// TIA Portal V20 program export: 3 tag tables, 2 data types, 2 data blocks, 7 code blocks (in call order from the OBs), 11 instance data blocks

VAR_GLOBAL   // PLC tag table "Default tag table"
   All_Lamps AT %QB0 : Byte;
   Lamps_On AT %Q5.0 : Bool;
   Light2State AT %M0.0 : Bool;
   Light1State AT %M0.1 : Bool;
   Light3State AT %M0.2 : Bool;
   LightStep AT %MW0 : Int;
   start AT %M2.0 : Bool;
   Elapsed_Time AT %MD4 : Time;
   Lamps AT %MB0 : Byte;
END_VAR

VAR_GLOBAL   // PLC tag table "Inputs"
   "Switch 1 ON" AT %I16.0 : Bool;
   "Switch 2 ON" AT %I16.1 : Bool;
   "Switch 3 ON" AT %I16.2 : Bool;
   "Switch 4 ON" AT %I16.3 : Bool;
   "Switch 5 ON" AT %I16.4 : Bool;
   "Switch 6 ON" AT %I16.5 : Bool;
   "Switch 7 ON" AT %I16.6 : Bool;
   "Switch 8 ON" AT %I16.7 : Bool;
   "Byte 1 ON" AT %IB1 : Byte;
   Here_is_a_word AT %IW2 : Word;
END_VAR

VAR_GLOBAL   // PLC tag table "Outputs"
   "Lamp 1 ON" AT %Q0.0 : Bool;
   "Lamp 2 ON" AT %Q0.1 : Bool;
   "Lamp 3 ON" AT %Q0.2 : Bool;
   "Lamp 4 ON" AT %Q0.3 : Bool;
   "Lamp 5 ON" AT %Q0.4 : Bool;
   "Lamp 6 ON" AT %Q0.5 : Bool;
   "Lamp 7 ON" AT %Q0.6 : Bool;
   "Lamp 8 ON" AT %Q0.7 : Bool;
   I_am_a_double_integer AT %QD1 : DInt;
END_VAR

TYPE "Equipment"
   STRUCT
      "type" : Int;
      commandOn : Bool;
      commandOff : Bool;
      feedbackOn : Bool;
      feedbackOff : Bool;
      isFaulty : Bool;
      isProcessFinished : Bool;
   END_STRUCT;
END_TYPE

TYPE "Tank"
   STRUCT
      isTankFull : Bool;
      tankLevel : Int;
      isEmpty : Bool;
      "type" : Bool;
   END_STRUCT;
END_TYPE

DATA_BLOCK "Global DB"   // DB7
{ S7_Optimized_Access := 'TRUE' }
// stored: MemoryReserve 100
   VAR
      Valve1 : "Equipment";
      Valve2 { S7_SetPoint := 'True'} : "Equipment";
      Valve3 { S7_SetPoint := 'True'} : "Equipment";
      Heater { S7_SetPoint := 'True'} : "Equipment";
      Mixer { S7_SetPoint := 'True'} : "Equipment";
      Process_Start { S7_SetPoint := 'True'} : Bool;
      Process_Stop : Bool;
      Process_Reset : Bool;
      Process_Step : Int;
      Process_Count : Int;
      isTankHeated : Bool;
      isTankMixed : Bool;
      Tank1 : "Tank";
      Tank2 { S7_SetPoint := 'True'} : "Tank";
      positive_edge { S7_SetPoint := 'True'} : Bool;
      prevLevel : DInt;
   END_VAR
BEGIN
   Heater."type" := 1;
   Mixer."type" := 2;
END_DATA_BLOCK

DATA_BLOCK "DB_Traffic_Lights"   // DB1
{ S7_Optimized_Access := 'TRUE' }
// stored: MemoryReserve 100
   VAR
      Process_Step : Int;
      Process_Start : Bool;
      "Timer" : IEC_TIMER;
      "Counter" { S7_SetPoint := 'True'} : IEC_COUNTER;
   END_VAR
   VAR RETAIN
      Positive_Edge { S7_SetPoint := 'True'} : Bool;
   END_VAR
   VAR
      Timer2 : IEC_TIMER;
   END_VAR
BEGIN
END_DATA_BLOCK

ORGANIZATION_BLOCK "Main"   // OB1, LAD, ProgramCycle
TITLE = "Main Program Sweep (Cycle)"
{ S7_Optimized_Access := 'TRUE' }
// stored: SetENOAutomatically false
   VAR_INPUT
      Initial_Call : Bool;   // Initial call of this OB
      Remanence : Bool;   // =True, if remanent data are available
   END_VAR
BEGIN

REGION Network 1
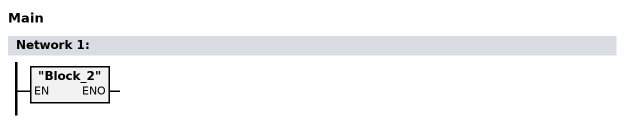
   RUNG wire#powerrail
      "Block_2"()
   END_RUNG
   // the same network as SCL:
   "Block_2"();
END_REGION
END_ORGANIZATION_BLOCK

FUNCTION "Block_2" : Void   // FC2, LAD
{ S7_Optimized_Access := 'TRUE' }
// stored: SetENOAutomatically false
   VAR_TEMP   // added for the SCL form of the ladder/FBD networks
      _w1 : Bool;
   END_VAR
BEGIN

REGION Network 1
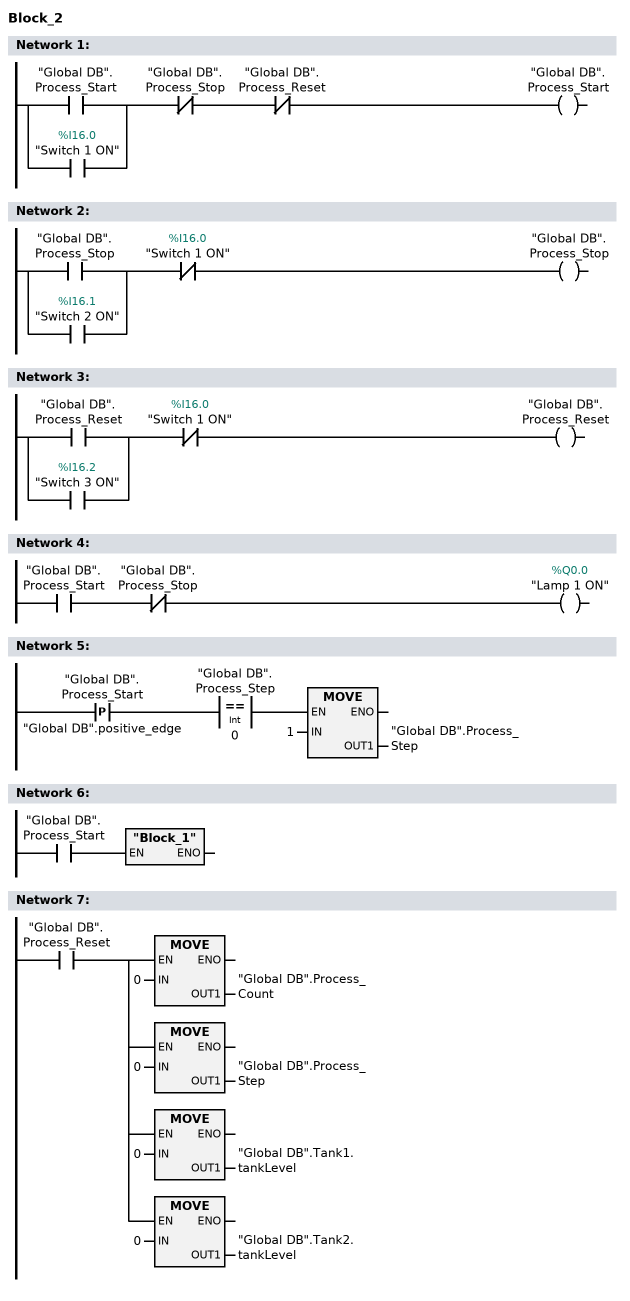
   RUNG wire#powerrail
      Contact( "Global DB".Process_Start )
      wire#w1
      I_Contact( "Global DB".Process_Stop )
      I_Contact( "Global DB".Process_Reset )
      Coil( "Global DB".Process_Start )
   END_RUNG
   RUNG wire#powerrail
      Contact( "Switch 1 ON" )
   END_RUNG wire#w1
   // the same network as SCL:
   "Global DB".Process_Start := ("Global DB".Process_Start OR "Switch 1 ON") AND NOT "Global DB".Process_Stop AND NOT "Global DB".Process_Reset;
END_REGION

REGION Network 2
   RUNG wire#powerrail
      Contact( "Global DB".Process_Stop )
      wire#w1
      I_Contact( "Switch 1 ON" )
      Coil( "Global DB".Process_Stop )
   END_RUNG
   RUNG wire#powerrail
      Contact( "Switch 2 ON" )
   END_RUNG wire#w1
   // the same network as SCL:
   "Global DB".Process_Stop := ("Global DB".Process_Stop OR "Switch 2 ON") AND NOT "Switch 1 ON";
END_REGION

REGION Network 3
   RUNG wire#powerrail
      Contact( "Global DB".Process_Reset )
      wire#w1
      I_Contact( "Switch 1 ON" )
      Coil( "Global DB".Process_Reset )
   END_RUNG
   RUNG wire#powerrail
      Contact( "Switch 3 ON" )
   END_RUNG wire#w1
   // the same network as SCL:
   "Global DB".Process_Reset := ("Global DB".Process_Reset OR "Switch 3 ON") AND NOT "Switch 1 ON";
END_REGION

REGION Network 4
   RUNG wire#powerrail
      Contact( "Global DB".Process_Start )
      I_Contact( "Global DB".Process_Stop )
      Coil( "Lamp 1 ON" )
   END_RUNG
   // the same network as SCL:
   "Lamp 1 ON" := "Global DB".Process_Start AND NOT "Global DB".Process_Stop;
END_REGION

REGION Network 5
   RUNG wire#powerrail
      P_Contact(operand := "Global DB".Process_Start, bit := "Global DB".positive_edge)
      { S7_Templates := "SrcType := Int" } EQ_Contact(in1 := "Global DB".Process_Step, in2 := 0)
      Move(in := 1, out1 => "Global DB".Process_Step)
   END_RUNG
   // the same network as SCL:
   #_w1 := "Global DB".Process_Start AND NOT "Global DB".positive_edge;   // rising edge of "Global DB".Process_Start
   "Global DB".positive_edge := "Global DB".Process_Start;
   IF #_w1 AND ("Global DB".Process_Step = 0) THEN "Global DB".Process_Step := 1; END_IF;
END_REGION

REGION Network 6
   RUNG wire#powerrail
      Contact( "Global DB".Process_Start )
      "Block_1"()
   END_RUNG
   // the same network as SCL:
   IF "Global DB".Process_Start THEN "Block_1"(); END_IF;
END_REGION

REGION Network 7
   RUNG wire#powerrail
      Contact( "Global DB".Process_Reset )
      wire#w1
      Move(in := 0, out1 => "Global DB".Process_Count)
   END_RUNG
   RUNG wire#w1
      Move(in := 0, out1 => "Global DB".Process_Step)
   END_RUNG
   RUNG wire#w1
      Move(in := 0, out1 => "Global DB".Tank1.tankLevel)
   END_RUNG
   RUNG wire#w1
      Move(in := 0, out1 => "Global DB".Tank2.tankLevel)
   END_RUNG
   // the same network as SCL:
   IF "Global DB".Process_Reset THEN
       "Global DB".Process_Count := 0;
       "Global DB".Process_Step := 0;
       "Global DB".Tank1.tankLevel := 0;
       "Global DB".Tank2.tankLevel := 0;
   END_IF;
END_REGION
END_FUNCTION

FUNCTION "Block_1" : Void
{ S7_Optimized_Access := 'TRUE' }
VERSION : 0.1
   VAR_TEMP 
      prevTankLevel : DInt;
   END_VAR


BEGIN
	
	CASE "Global DB".Process_Step OF
	        
	    1:
	        
	        "Block_3"(eqp := "Global DB".Valve1,
	                  timer := "IEC_Timer_0_DB_4",
	                  tank := "Global DB".Tank1);
	      
	        
	        ;
	        
	        
	    2:
	        
	        "Block_3"(eqp := "Global DB".Heater,
	                  timer := "IEC_Timer_0_DB_5",
	                  tank := "Global DB".Tank1);
	        ;
	        
	        
	    3:
	        "Block_3"(eqp := "Global DB".Mixer,
	                  timer := "IEC_Timer_0_DB_6",
	                  tank := "Global DB".Tank1);
	        ;
	        
	        
	    4:
	 
	        IF ("Global DB".Process_Count < 5) THEN
	            
	            
	            
	            "Global DB".Tank2.tankLevel := "Global DB".prevLevel + (DINT_TO_REAL(TIME_TO_DINT("IEC_Timer_0_DB_7".ET)) / 250.0);
	            "Global DB".Tank1.tankLevel := 100 - DINT_TO_REAL(TIME_TO_DINT("IEC_Timer_0_DB_7".ET)) / 50.0;
	            
	            
	            IF ("IEC_Timer_0_DB_7".Q) THEN
	                
	                
	                "Global DB".prevLevel := "Global DB".Tank2.tankLevel;
	                IF ("Global DB".Tank2.isTankFull) THEN
	                    "Global DB".Process_Step := 5;
	                    "Global DB".Process_Count := 0;
	                ELSE
	                    "Global DB".Process_Count += 1;
	                    "Global DB".Process_Step := 1;
	                END_IF;
	                
	            END_IF;
	            
	            
	        END_IF;
	        
	     5:
	
	         "Global DB".Tank2.tankLevel := 100 - DINT_TO_REAL(TIME_TO_DINT("IEC_Timer_0_DB_8".ET))/ 50.0;
	         
	         IF("IEC_Timer_0_DB_8".Q) THEN
	         "Global DB".Process_Step := 1;
	         "Global DB".prevLevel := 0;
	         
	        END_IF
	         
	         ;
	        
	        
	        
	END_CASE;
	
	"IEC_Timer_0_DB_7".TON(IN := "Global DB".Process_Step = 4,
	                       PT := T#5s);
	
	"IEC_Timer_0_DB_8".TON(IN := "Global DB".Process_Step = 5,
	                       PT := T#5s);
	
	IF ("Global DB".Tank1.tankLevel = 100) THEN
	    "Global DB".Tank1.isTankFull := TRUE
	    ;
	ELSE
	    "Global DB".Tank1.isTankFull := FALSE;
	    
	END_IF;
	
	IF ("Global DB".Tank2.tankLevel = 100) THEN
	    "Global DB".Tank2.isTankFull := TRUE
	    ;
	ELSE
	    "Global DB".Tank2.isTankFull := FALSE;
	    
	END_IF;
END_FUNCTION

FUNCTION "Block_3" : Void
{ S7_Optimized_Access := 'TRUE' }
VERSION : 0.1
   VAR_IN_OUT 
      eqp : "Equipment";
      "timer" {InstructionName := 'IEC_TIMER'; LibVersion := '1.0'} : IEC_TIMER;
      tank : "Tank";
   END_VAR

   VAR_TEMP 
      isNotTank : Bool;
      currentStep : Int;
      currentStepOld : Int;
      isStepDifferent : Bool;
   END_VAR


BEGIN
	
	#eqp.commandOn := TRUE;
	
	
	    
	"IEC_Timer_0_DB_4".TON(
	                       IN := ("Global DB".Process_Step = 1),
	                       PT := T#5s
	                       
	);
	
	"IEC_Timer_0_DB_5".TON(
	                       IN := ("Global DB".Process_Step = 2),
	                       PT := T#5s
	                       
	);
	
	
	
	
	
	
	"IEC_Timer_0_DB_6".TON(
	                       IN := ("Global DB".Process_Step = 3),
	                       PT := T#5s
	                       
	);
	
	
	  
	    CASE #eqp.type OF
	        0:
	            #tank.tankLevel := DINT_TO_REAL(TIME_TO_DINT(#timer.ET)) / 50.0;
	            
	        1..2:
	            #eqp.isProcessFinished := TRUE;
	            
	            
	    END_CASE;
	    
	
	    IF ( #timer.Q) THEN
	        #eqp.commandOn := FALSE;
	        #eqp.commandOff := TRUE;
	        "Global DB".Process_Step += 1
	        ;
	    END_IF;
	    
	 
END_FUNCTION

FUNCTION_BLOCK "FC_Traffic_Lights"   // FB1, LAD
{ S7_Optimized_Access := 'TRUE' }
// stored: MemoryReserve 100, SetENOAutomatically false
   VAR
      "Timer" { S7_SetPoint := 'True'} : TON_TIME;
   END_VAR
   VAR_TEMP   // added for the SCL form of the ladder/FBD networks
      _w1 : Bool;
   END_VAR
BEGIN

REGION Network 1
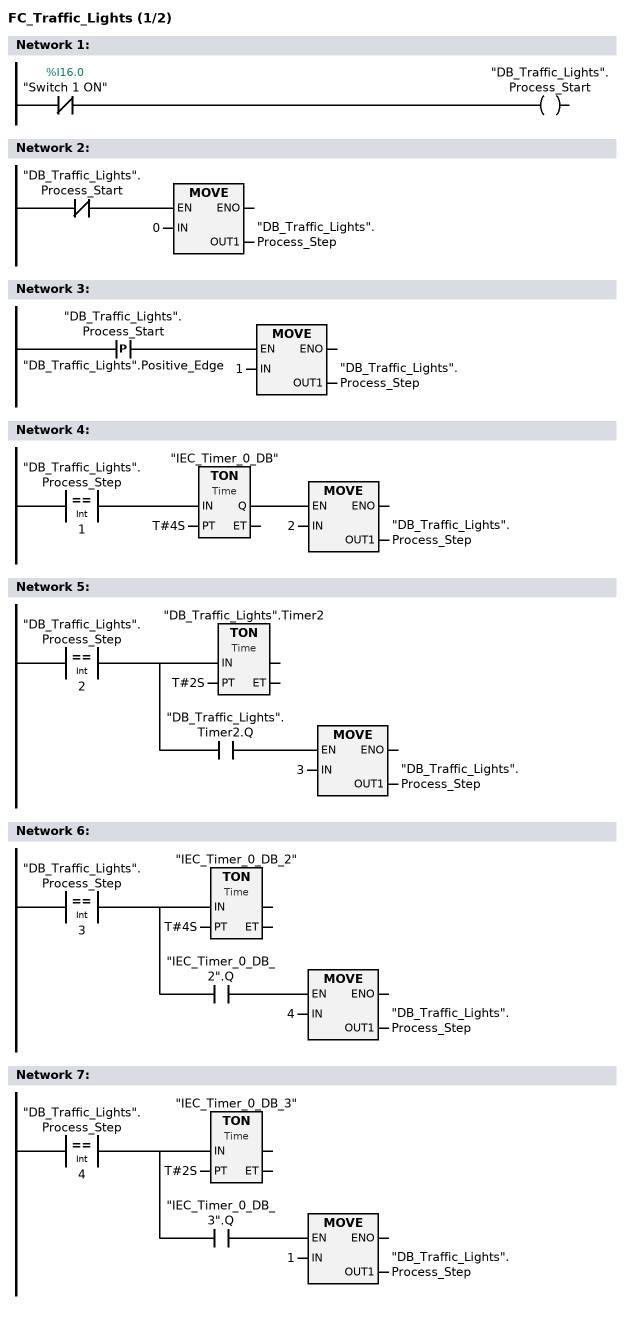
   RUNG wire#powerrail
      I_Contact( "Switch 1 ON" )
      Coil( "DB_Traffic_Lights".Process_Start )
   END_RUNG
   // the same network as SCL:
   "DB_Traffic_Lights".Process_Start := NOT "Switch 1 ON";
END_REGION

REGION Network 2
   RUNG wire#powerrail
      I_Contact( "DB_Traffic_Lights".Process_Start )
      Move(in := 0, out1 => "DB_Traffic_Lights".Process_Step)
   END_RUNG
   // the same network as SCL:
   IF NOT "DB_Traffic_Lights".Process_Start THEN "DB_Traffic_Lights".Process_Step := 0; END_IF;
END_REGION

REGION Network 3
   RUNG wire#powerrail
      P_Contact(operand := "DB_Traffic_Lights".Process_Start, bit := "DB_Traffic_Lights".Positive_Edge)
      Move(in := 1, out1 => "DB_Traffic_Lights".Process_Step)
   END_RUNG
   // the same network as SCL:
   #_w1 := "DB_Traffic_Lights".Process_Start AND NOT "DB_Traffic_Lights".Positive_Edge;   // rising edge of "DB_Traffic_Lights".Process_Start
   "DB_Traffic_Lights".Positive_Edge := "DB_Traffic_Lights".Process_Start;
   IF #_w1 THEN "DB_Traffic_Lights".Process_Step := 1; END_IF;
END_REGION

REGION Network 4
   RUNG wire#powerrail
      { S7_Templates := "SrcType := Int" } EQ_Contact(in1 := "DB_Traffic_Lights".Process_Step, in2 := 1)
      { S7_Templates := "time_type := Time" } "IEC_Timer_0_DB".TON(pt := T#4S, et =>)
      Move(in := 2, out1 => "DB_Traffic_Lights".Process_Step)
   END_RUNG
   // the same network as SCL:
   "IEC_Timer_0_DB".TON(IN := "DB_Traffic_Lights".Process_Step = 1, PT := T#4S);
   IF "IEC_Timer_0_DB".Q THEN "DB_Traffic_Lights".Process_Step := 2; END_IF;
END_REGION

REGION Network 5
   RUNG wire#powerrail
      { S7_Templates := "SrcType := Int" } EQ_Contact(in1 := "DB_Traffic_Lights".Process_Step, in2 := 2)
      wire#w1
      { S7_Templates := "time_type := Time" } "DB_Traffic_Lights".Timer2.TON(pt := T#2S, et =>)
   END_RUNG
   RUNG wire#w1
      Contact( "DB_Traffic_Lights".Timer2.Q )
      Move(in := 3, out1 => "DB_Traffic_Lights".Process_Step)
   END_RUNG
   // the same network as SCL:
   #_w1 := "DB_Traffic_Lights".Process_Step = 2;
   "DB_Traffic_Lights".Timer2.TON(IN := #_w1, PT := T#2S);
   IF #_w1 AND "DB_Traffic_Lights".Timer2.Q THEN "DB_Traffic_Lights".Process_Step := 3; END_IF;
END_REGION

REGION Network 6
   RUNG wire#powerrail
      { S7_Templates := "SrcType := Int" } EQ_Contact(in1 := "DB_Traffic_Lights".Process_Step, in2 := 3)
      wire#w1
      { S7_Templates := "time_type := Time" } "IEC_Timer_0_DB_2".TON(pt := T#4S, et =>)
   END_RUNG
   RUNG wire#w1
      Contact( "IEC_Timer_0_DB_2".Q )
      Move(in := 4, out1 => "DB_Traffic_Lights".Process_Step)
   END_RUNG
   // the same network as SCL:
   #_w1 := "DB_Traffic_Lights".Process_Step = 3;
   "IEC_Timer_0_DB_2".TON(IN := #_w1, PT := T#4S);
   IF #_w1 AND "IEC_Timer_0_DB_2".Q THEN "DB_Traffic_Lights".Process_Step := 4; END_IF;
END_REGION

REGION Network 7
   RUNG wire#powerrail
      { S7_Templates := "SrcType := Int" } EQ_Contact(in1 := "DB_Traffic_Lights".Process_Step, in2 := 4)
      wire#w1
      { S7_Templates := "time_type := Time" } "IEC_Timer_0_DB_3".TON(pt := T#2S, et =>)
   END_RUNG
   RUNG wire#w1
      Contact( "IEC_Timer_0_DB_3".Q )
      Move(in := 1, out1 => "DB_Traffic_Lights".Process_Step)
   END_RUNG
   // the same network as SCL:
   #_w1 := "DB_Traffic_Lights".Process_Step = 4;
   "IEC_Timer_0_DB_3".TON(IN := #_w1, PT := T#2S);
   IF #_w1 AND "IEC_Timer_0_DB_3".Q THEN "DB_Traffic_Lights".Process_Step := 1; END_IF;
END_REGION

REGION Network 8: Step
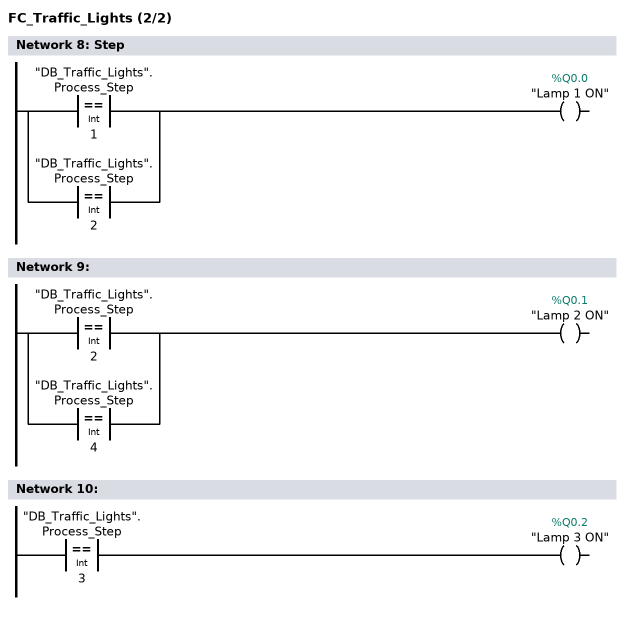
   RUNG wire#powerrail
      { S7_Templates := "SrcType := Int" } EQ_Contact(in1 := "DB_Traffic_Lights".Process_Step, in2 := 1)
      wire#w1
      Coil( "Lamp 1 ON" )
   END_RUNG
   RUNG wire#powerrail
      { S7_Templates := "SrcType := Int" } EQ_Contact(in1 := "DB_Traffic_Lights".Process_Step, in2 := 2)
   END_RUNG wire#w1
   // the same network as SCL:
   "Lamp 1 ON" := ("DB_Traffic_Lights".Process_Step = 1) OR ("DB_Traffic_Lights".Process_Step = 2);
END_REGION

REGION Network 9
   RUNG wire#powerrail
      { S7_Templates := "SrcType := Int" } EQ_Contact(in1 := "DB_Traffic_Lights".Process_Step, in2 := 2)
      wire#w1
      Coil( "Lamp 2 ON" )
   END_RUNG
   RUNG wire#powerrail
      { S7_Templates := "SrcType := Int" } EQ_Contact(in1 := "DB_Traffic_Lights".Process_Step, in2 := 4)
   END_RUNG wire#w1
   // the same network as SCL:
   "Lamp 2 ON" := ("DB_Traffic_Lights".Process_Step = 2) OR ("DB_Traffic_Lights".Process_Step = 4);
END_REGION

REGION Network 10
   RUNG wire#powerrail
      { S7_Templates := "SrcType := Int" } EQ_Contact(in1 := "DB_Traffic_Lights".Process_Step, in2 := 3)
      Coil( "Lamp 3 ON" )
   END_RUNG
   // the same network as SCL:
   "Lamp 3 ON" := "DB_Traffic_Lights".Process_Step = 3;
END_REGION
END_FUNCTION_BLOCK

FUNCTION "Block_4" : Void   // FC4, STL
{ S7_Optimized_Access := 'TRUE' }
BEGIN

NETWORK
TITLE = 
      A     "Switch 1 ON";
      =     "Lamp 1 ON";
END_FUNCTION

FUNCTION "Block_5" : Void   // FC5, FBD
{ S7_Optimized_Access := 'TRUE' }
// stored: SetENOAutomatically false
BEGIN

REGION Network 1
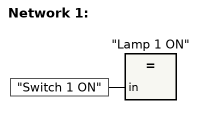
   "Lamp 1 ON" := "Switch 1 ON";
END_REGION
END_FUNCTION

DATA_BLOCK "FC_Traffic_Lights_DB"   // DB3
// stored: InstanceOfName FC_Traffic_Lights, InstanceOfType FB
"FC_Traffic_Lights"
BEGIN
END_DATA_BLOCK

DATA_BLOCK "FC_Traffic_Lights_DB_1"   // DB9
// stored: InstanceOfName FC_Traffic_Lights, InstanceOfType FB
"FC_Traffic_Lights"
BEGIN
END_DATA_BLOCK

DATA_BLOCK "IEC_Timer_0_DB"   // DB4
{ S7_Optimized_Access := 'TRUE' }
// stored: InstanceOfName IEC_TIMER, OfSystemLibElement IEC_TIMER, OfSystemLibVersion 1.0
"IEC_TIMER"
   // VAR
   //    PT : Time;
   //    ET { ExternalWritable := 'False'} : Time;
   //    IN : Bool;
   //    Q { ExternalWritable := 'False'} : Bool;
   // END_VAR
BEGIN
END_DATA_BLOCK

DATA_BLOCK "IEC_Timer_0_DB_1"   // DB2
{ S7_Optimized_Access := 'TRUE' }
// stored: InstanceOfName IEC_TIMER, OfSystemLibElement IEC_TIMER, OfSystemLibVersion 1.0
"IEC_TIMER"
   // VAR
   //    PT : Time;
   //    ET { ExternalWritable := 'False'} : Time;
   //    IN : Bool := true;
   //    Q { ExternalWritable := 'False'} : Bool;
   // END_VAR
BEGIN
END_DATA_BLOCK

DATA_BLOCK "IEC_Timer_0_DB_2"   // DB5
{ S7_Optimized_Access := 'TRUE' }
// stored: InstanceOfName IEC_TIMER, OfSystemLibElement IEC_TIMER, OfSystemLibVersion 1.0
"IEC_TIMER"
   // VAR
   //    PT : Time;
   //    ET { ExternalWritable := 'False'} : Time;
   //    IN : Bool;
   //    Q { ExternalWritable := 'False'} : Bool;
   // END_VAR
BEGIN
END_DATA_BLOCK

DATA_BLOCK "IEC_Timer_0_DB_3"   // DB6
{ S7_Optimized_Access := 'TRUE' }
// stored: InstanceOfName IEC_TIMER, OfSystemLibElement IEC_TIMER, OfSystemLibVersion 1.0
"IEC_TIMER"
   // VAR
   //    PT : Time;
   //    ET { ExternalWritable := 'False'} : Time;
   //    IN : Bool;
   //    Q { ExternalWritable := 'False'} : Bool;
   // END_VAR
BEGIN
END_DATA_BLOCK

DATA_BLOCK "IEC_Timer_0_DB_4"   // DB8
{ S7_Optimized_Access := 'TRUE' }
// stored: AutoNumber false, InstanceOfName IEC_TIMER, OfSystemLibElement IEC_TIMER, OfSystemLibVersion 1.0
"IEC_TIMER"
   // VAR
   //    PT : Time;
   //    ET { ExternalWritable := 'False'} : Time;
   //    IN : Bool;
   //    Q { ExternalWritable := 'False'} : Bool;
   // END_VAR
BEGIN
END_DATA_BLOCK

DATA_BLOCK "IEC_Timer_0_DB_5"   // DB10
{ S7_Optimized_Access := 'TRUE' }
// stored: InstanceOfName IEC_TIMER, OfSystemLibElement IEC_TIMER, OfSystemLibVersion 1.0
"IEC_TIMER"
   // VAR
   //    PT : Time;
   //    ET { ExternalWritable := 'False'} : Time;
   //    IN : Bool;
   //    Q { ExternalWritable := 'False'} : Bool;
   // END_VAR
BEGIN
END_DATA_BLOCK

DATA_BLOCK "IEC_Timer_0_DB_6"   // DB11
{ S7_Optimized_Access := 'TRUE' }
// stored: InstanceOfName IEC_TIMER, OfSystemLibElement IEC_TIMER, OfSystemLibVersion 1.0
"IEC_TIMER"
   // VAR
   //    PT : Time;
   //    ET { ExternalWritable := 'False'} : Time;
   //    IN : Bool;
   //    Q { ExternalWritable := 'False'} : Bool;
   // END_VAR
BEGIN
END_DATA_BLOCK

DATA_BLOCK "IEC_Timer_0_DB_7"   // DB12
{ S7_Optimized_Access := 'TRUE' }
// stored: InstanceOfName IEC_TIMER, OfSystemLibElement IEC_TIMER, OfSystemLibVersion 1.0
"IEC_TIMER"
   // VAR
   //    PT : Time;
   //    ET { ExternalWritable := 'False'} : Time;
   //    IN : Bool;
   //    Q { ExternalWritable := 'False'} : Bool;
   // END_VAR
BEGIN
END_DATA_BLOCK

DATA_BLOCK "IEC_Timer_0_DB_8"   // DB13
{ S7_Optimized_Access := 'TRUE' }
// stored: InstanceOfName IEC_TIMER, OfSystemLibElement IEC_TIMER, OfSystemLibVersion 1.0
"IEC_TIMER"
   // VAR
   //    PT : Time;
   //    ET { ExternalWritable := 'False'} : Time;
   //    IN : Bool;
   //    Q { ExternalWritable := 'False'} : Bool;
   // END_VAR
BEGIN
END_DATA_BLOCK
